(* IEC 61131-3 sources: volt/packages/volt-lsp-iec/test-corpus/lenze-mid/Device/Plc Logic/Application/Library Manager/(unresolved)/cmpopcuaserver interfaces, 18 files *)

(* ---- EVTPARAM_CMPOPCUASERVERSESSIONSCHANGED.dut ---- *)
TYPE EVTPARAM_CMPOPCUASERVERSESSIONSCHANGED :
STRUCT
	EVENT : OpcUaServer_SessionEvents;
	DWSESSIONID : DWORD;
END_STRUCT
END_TYPE

(* ---- OPCUADATATYPEDESCRIPTION.dut ---- *)
TYPE OPCUADATATYPEDESCRIPTION :
STRUCT
	ISABSTRACT : OpcUa_Boolean;
	BDATATYPEDEFINITIONSET : OpcUa_Boolean;
	DATATYPEDEFINITION : OpcUa_ExtensionObject;
END_STRUCT
END_TYPE

(* ---- OPCUAELEMENTDESCRIPTION.dut ---- *)
TYPE OPCUAELEMENTDESCRIPTION :
UNION
	OBJECT : OpcUaObjectDescription;
	VARIABLE : OpcUaVariableDescription;
	UAMETHOD : OpcUaMethodDescription;
	OBJECTTYPE : OpcUaObjectTypeDescription;
	VARIABLETYPE : OpcUaVariableTypeDescription;
	REFERENCETYPE : OpcUaReferenceTypeDescription;
	DATATYPE : OpcUaDataTypeDescription;
	VIEW : OpcUaViewDescription;
END_UNION
END_TYPE

(* ---- OPCUAMETHODDESCRIPTION.dut ---- *)
TYPE OPCUAMETHODDESCRIPTION :
STRUCT
	EXECUTABLE : OpcUa_Boolean;
	USEREXECUTABLE : OpcUa_Boolean;
END_STRUCT
END_TYPE

(* ---- OPCUAOBJECTDESCRIPTION.dut ---- *)
TYPE OPCUAOBJECTDESCRIPTION :
STRUCT
	EVENTNOTIFIER : OpcUa_Byte;
END_STRUCT
END_TYPE

(* ---- OPCUAOBJECTTYPEDESCRIPTION.dut ---- *)
TYPE OPCUAOBJECTTYPEDESCRIPTION :
STRUCT
	ISABSTRACT : OpcUa_Boolean;
END_STRUCT
END_TYPE

(* ---- OPCUAREFERENCETYPEDESCRIPTION.dut ---- *)
TYPE OPCUAREFERENCETYPEDESCRIPTION :
STRUCT
	ISABSTRACT : OpcUa_Boolean;
	SYMMETRIC : OpcUa_Boolean;
	BINVERSENAMESET : OpcUa_Boolean;
	INVERSENAME : OpcUa_LocalizedText;
END_STRUCT
END_TYPE

(* ---- OPCUASERVER_BROWSEPATH.dut ---- *)
TYPE OPCUASERVER_BROWSEPATH :
STRUCT
	UI32NUMOFELEMENTS : OpcUa_UInt32;
	PBROWSEPATH : POINTER TO OpcUa_QualifiedName;
END_STRUCT
END_TYPE

(* ---- OPCUASERVER_MESSAGESECURITYMODE.dut ---- *)
TYPE OPCUASERVER_MESSAGESECURITYMODE :
(
	INVALID := 0,
	NONE,
	SIGN,
	SIGNANDENCRYPT
);
END_TYPE

(* ---- OPCUASERVER_SESSION_INFORMATION.dut ---- *)
TYPE OPCUASERVER_SESSION_INFORMATION :
STRUCT
	DWSESSIONID : DWORD;
	CLIENTADDRESS : INADDR;
	PWSSESSIONNAME : WSTRING(255);
	PWSAPPLICATIONNAME : WSTRING(255);
	PWSAPPLICATIONURI : WSTRING(255);
	PWSPRODUCTURI : WSTRING(255);
	PWSSECURITYPOLICY : WSTRING(255);
	SECURITYMODE : OpcUaServer_MessageSecurityMode;
	HCLIENTCERTIFICATE : RTS_IEC_HANDLE;
	HUSER : RTS_IEC_HANDLE;
END_STRUCT
END_TYPE

(* ---- OPCUASERVER_SESSIONEVENTS.dut ---- *)
TYPE OPCUASERVER_SESSIONEVENTS :
(
	SESSION_ADDED := 1,
	SESSION_CHANGED,
	SESSION_REMOVED
);
END_TYPE

(* ---- OPCUASERVEREVENTFIELD.dut ---- *)
TYPE OPCUASERVEREVENTFIELD :
STRUCT
	PATH : OpcUaServer_BrowsePath;
	VALUE : OpcUa_Variant;
	ATTRIBUTEID : OpcUa_UInt32;
END_STRUCT
END_TYPE

(* ---- OPCUASERVERNODEDESCRIPTION.dut ---- *)
TYPE OPCUASERVERNODEDESCRIPTION :
STRUCT
	NODEID : OpcUa_NodeId;
	NODECLASS : OpcUa_NodeClass;
	BROWSENAME : OpcUa_QualifiedName;
	DISPLAYNAME : OpcUa_LocalizedText;
	BDESCRIPTIONSET : OpcUa_Boolean;
	DESCRIPTION : OpcUa_LocalizedText;
	BWRITEMASKSET : OpcUa_Boolean;
	UI32WRITEMASK : OpcUa_UInt32;
	BUSERWRITEMASKSET : OpcUa_Boolean;
	UI32USERWRITEMASK : OpcUa_UInt32;
	BACCESSRESTRICTIONSSET : OpcUa_Boolean;
	UI16ACCESSRESTRICTIONS : OpcUa_UInt16;
	BROLEPERMISSIONSSET : OpcUa_Boolean;
	ROLEPERMISSIONS : OpcUa_Variant;
	BUSERROLEPERMISSIONSSET : OpcUa_Boolean;
	USERROLEPERMISSIONS : OpcUa_Variant;
	TYPEDEFINITION : OpcUa_NodeId;
	ELEMENTDESCRIPTION : OpcUaElementDescription;
	PSZOBJECT : POINTER TO STRING;
END_STRUCT
END_TYPE

(* ---- OPCUASERVERREFERENCEDESCRIPTION.dut ---- *)
TYPE OPCUASERVERREFERENCEDESCRIPTION :
STRUCT
	STARTNODE : OpcUa_NodeId;
	DESTINATIONNODE : OpcUa_NodeId;
	REFERENCETYPE : OpcUa_NodeId;
	BBIDIRECTIONAL : OpcUa_Boolean;
END_STRUCT
END_TYPE

(* ---- OPCUAVARIABLEDESCRIPTION.dut ---- *)
TYPE OPCUAVARIABLEDESCRIPTION :
STRUCT
	BVALUEAVAILABLE : OpcUa_Boolean;
	VALUE : OpcUa_Variant;
	DATATYPE : OpcUa_NodeId;
	I32VALUERANK : OpcUa_Int32;
	ACCESSLEVEL : OpcUa_Byte;
	USERACCESSLEVEL : OpcUa_Byte;
	HISTORIZING : OpcUa_Boolean;
	BARRAYDIMENSIONSET : OpcUa_Boolean;
	ARRAYDIMENSIONS : OpcUa_Variant;
	BMINIMUMSAMPLINGINTERVALSET : OpcUa_Boolean;
	MINIMUMSAMPLINGINTERVAL : OpcUa_Double;
	BACCESSLEVELEXSET : OpcUa_Boolean;
	UI32ACCESSLEVELEX : OpcUa_UInt32;
END_STRUCT
END_TYPE

(* ---- OPCUAVARIABLETYPEDESCRIPTION.dut ---- *)
TYPE OPCUAVARIABLETYPEDESCRIPTION :
STRUCT
	DATATYPE : OpcUa_NodeId;
	I32VALUERANK : OpcUa_Int32;
	ISABSTRACT : OpcUa_Boolean;
	BVALUESET : OpcUa_Boolean;
	VALUE : OpcUa_Variant;
	BARRAYDIMENSIONSSET : OpcUa_Boolean;
	ARRAYDIMENSIONS : OpcUa_Variant;
END_STRUCT
END_TYPE

(* ---- OPCUAVIEWDESCRIPTION.dut ---- *)
TYPE OPCUAVIEWDESCRIPTION :
STRUCT
	CONTAINSNOLOOPS : OpcUa_Boolean;
	EVENTNOTIFIER : OpcUa_Byte;
END_STRUCT
END_TYPE

(* ---- EVENTIDS.gvl ---- *)
VAR_GLOBAL
	CMPID_CMPOPCUASERVER : DWORD := 16#124;
	EVTPARAMID_CMPOPCUASERVERSESSIONSCHANGED : WORD := 16#1;
	EVTVERSION_CMPOPCUASERVERSESSIONSCHANGED : WORD := 16#1;
	EVT_CMPOPCUASERVERSESSIONSCHANGED : DWORD := (SHL(UINT_TO_DWORD(EventClass.EVTCLASS_INFO), 16) OR 16#1);
END_VAR
